FUNCTION_BLOCK FB_Blink   //脉冲发生器
VAR_INPUT
	EN:			BOOL;
	Intervall:		TIME;
END_VAR
VAR_OUTPUT
	Blink:		BOOL;
END_VAR
VAR
	TON_01:		TON;
	TON_02:		TON;
END_VAR

IF EN THEN
	TON_01	(IN:=	NOT TON_02.Q, PT:=Intervall);
	TON_02	(IN:=	 TON_01.Q, PT:=Intervall);
	Blink:= TON_01.Q;
ELSE
	Blink := FALSE;
END_IF

END_FUNCTION_BLOCK

(* stored: Version 1.1.0.1, ProductVersion 3.1.4024.9
   POU FB_Blink: Id {4566fe1d-59b4-4a08-adcb-d7e555dde4ff}, SpecialFunc None *)
